(* PLC project speed, Dassault Systèmes ControlBuild 2024x *)
(* stored: creationDateTime 2023-10-03T11:13:50-01:00 *)

FUNCTION_BLOCK tni_train.speed
  VAR_OUTPUT
    speed : REAL := 0.0;
  END_VAR


END_FUNCTION_BLOCK
